// TIA Portal V20 export
TYPE "typeSequenceControlNodeJobInterface"
// stored: Namespace Unit1.Em5
   STRUCT
      commands { ExternalWritable := 'False'} : "Unit1.Em5.typeSequenceControlNodeJobInterfaceCommands";
      monitoring { ExternalWritable := 'False'} : "Unit1.Em5.typeSequenceControlNodeJobInterfaceMonitoring";
   END_STRUCT;
END_TYPE
